// Represents the seconds of the current minute, ranging from 0 to 59.
TYPE T_Second : UINT(0..59); END_TYPE

(* stored: Version 1.1.0.1
   DUT T_Second: Id {c5f44eb4-e975-0361-06dc-1cc66b18d41e} *)
